// TIA Portal V20 export
TYPE "type_emRelations_em2_sequence"
// stored: Access Published, Namespace Unit1
   STRUCT
      jrOutPnPLeft : Struct
         jobs : "LAF_typeJobs";
         sequence : "LAF_typeSequence";
         selectJobStatus { S7_SetPoint := 'True'} : Array[0..10] of "LAF_typeJobStatus";
         "step" : "LER_typeStep";
         jobInterface : Struct
            stack1LoadJob2 : "LER_typeJobInterface";
            stack2LoadJob3 : "LER_typeJobInterface";
            unloadJob4 : "LER_typeJobInterface";
         END_STRUCT;
         homeCheck : Struct
            partNoDetect { ExternalWritable := 'False'} : Bool;
            partDetect { ExternalWritable := 'False'} : Bool;
         END_STRUCT;
      END_STRUCT;
      jrOutPnPRight : Struct
         jobs : "LAF_typeJobs";
         sequence : "LAF_typeSequence";
         selectJobStatus { S7_SetPoint := 'True'} : Array[0..10] of "LAF_typeJobStatus";
         "step" : "LER_typeStep";
         jobInterface : Struct
            loadJob2 : "LER_typeJobInterface";
            unloadJob3 : "LER_typeJobInterface";
         END_STRUCT;
         homeCheck : Struct
            partNoDetect { ExternalWritable := 'False'} : Bool;
            partDetect { ExternalWritable := 'False'} : Bool;
         END_STRUCT;
      END_STRUCT;
   END_STRUCT;
   // // jrOutPnPLeft."step".action1[101] : Step[101] : JOB[1] Condition
   // // jrOutPnPLeft."step".action1[110] : Step[110] : JR PP Left Clamp Open
   // // jrOutPnPLeft."step".action1[130] : Step[130] : JR PP Left Clamp Close
   // // jrOutPnPLeft."step".action1[170] : Step[170] : JR PP Left Z-Axis Wait Pos
   // // jrOutPnPLeft."step".action1[180] : Step[180] : JR PP Left X-Axis Wait Pos
   // // jrOutPnPLeft."step".action1[190] : Step[190] : JOB[1] Step End
   // // jrOutPnPLeft."step".action1[201] : Step[201] : JOB[2] Condition
   // // jrOutPnPLeft."step".action1[210] : Step[210] : JR PP Left X-Axis Loading Pos[Stack-1]
   // // jrOutPnPLeft."step".action1[211] : Step[211] : JR PP Left Z-Axis Loading Pos[Stack-1]
   // // jrOutPnPLeft."step".action1[220] : Step[220] : JR PP Left [OnPosition Unloading] => Stack #1
   // // jrOutPnPLeft."step".action1[221] : Step[221] : JR PP Left Clamp Close
   // // jrOutPnPLeft."step".action1[222] : Step[222] : JR PP Left [Request Unclamp] => Stack #1
   // // jrOutPnPLeft."step".action1[280] : Step[280] : JR PP Left X/Z-Axis Wait Pos
   // // jrOutPnPLeft."step".action1[290] : Step[290] : JOB[2] Step End
   // // jrOutPnPLeft."step".action1[301] : Step[301] : JOB[3] Condition
   // // jrOutPnPLeft."step".action1[310] : Step[310] : JR PP Left X-Axis Loading Pos[Stack-2]
   // // jrOutPnPLeft."step".action1[311] : Step[311] : JR PP left Z-Axis Loading Pos[Stack-2]
   // // jrOutPnPLeft."step".action1[320] : Step[320] : JR PP Left [OnPosition Unloading] => Stack #2
   // // jrOutPnPLeft."step".action1[321] : Step[321] : JR PP Left Clamp Close
   // // jrOutPnPLeft."step".action1[322] : Step[322] : JR PP Left [Request Unclamp] => Stack #2
   // // jrOutPnPLeft."step".action1[380] : Step[380] : JR PP Left X/Z-Axis Wait Pos
   // // jrOutPnPLeft."step".action1[390] : Step[390] : JOB[3] Step End
   // // jrOutPnPLeft."step".action1[401] : Step[401] : JOB[4] Condition
   // // jrOutPnPLeft."step".action1[410] : Step[410] : JR PP Left X-Axis Put Pos
   // // jrOutPnPLeft."step".action1[411] : Step[411] : JR PP Left Z-Axis Put Pos
   // // jrOutPnPLeft."step".action1[420] : Step[420] : JR PP Left [Unloading Ready] => Top Tape Fix Stage
   // // jrOutPnPLeft."step".action1[421] : Step[421] : JR PP Left Clamp Open
   // // jrOutPnPLeft."step".action1[422] : Step[422] : JR PP Left [Unclamp Done] => Top Tape Fix Stage
   // // jrOutPnPLeft."step".action1[480] : Step[480] : JR PP Left X/Z-Axis Wait Pos
   // // jrOutPnPLeft."step".action1[490] : Step[490] : JOB[4] Step End
   // // jrOutPnPLeft."step".transition1[101] : Step[101] : JOB[1] Condition
   // // jrOutPnPLeft."step".transition1[110] : Step[110] : JR PP Left Clamp Open
   // // jrOutPnPLeft."step".transition1[130] : Step[130] : JR PP Left Clamp Close
   // // jrOutPnPLeft."step".transition1[170] : Step[170] : JR PP Left Z-Axis Wait Pos
   // // jrOutPnPLeft."step".transition1[180] : Step[180] : JR PP Left X-Axis Wait Pos
   // // jrOutPnPLeft."step".transition1[190] : Step[190] : JOB[1] Step End
   // // jrOutPnPLeft."step".transition1[201] : Step[201] : JOB[2] Condition
   // // jrOutPnPLeft."step".transition1[210] : Step[210] : JR PP Left X-Axis Loading Pos[Stack-1]
   // // jrOutPnPLeft."step".transition1[211] : Step[211] : JR PP Left Z-Axis Loading Pos[Stack-1]
   // // jrOutPnPLeft."step".transition1[220] : Step[220] : JR PP Left [OnPosition Unloading] => Stack #1
   // // jrOutPnPLeft."step".transition1[221] : Step[221] : JR PP Left Clamp Close
   // // jrOutPnPLeft."step".transition1[222] : Step[222] : JR PP Left [Request Unclamp] => Stack #1
   // // jrOutPnPLeft."step".transition1[280] : Step[280] : JR PP Left X/Z-Axis Wait Pos
   // // jrOutPnPLeft."step".transition1[290] : Step[290] : JOB[2] Step End
   // // jrOutPnPLeft."step".transition1[301] : Step[301] : JOB[3] Condition
   // // jrOutPnPLeft."step".transition1[310] : Step[310] : JR PP Left X-Axis Loading Pos[Stack-2]
   // // jrOutPnPLeft."step".transition1[311] : Step[311] : JR PP left Z-Axis Loading Pos[Stack-2]
   // // jrOutPnPLeft."step".transition1[320] : Step[320] : JR PP Left [OnPosition Unloading] => Stack #2
   // // jrOutPnPLeft."step".transition1[321] : Step[321] : JR PP Left Clamp Close
   // // jrOutPnPLeft."step".transition1[322] : Step[322] : JR PP Left [Request Unclamp] => Stack #2
   // // jrOutPnPLeft."step".transition1[380] : Step[380] : JR PP Left X/Z-Axis Wait Pos
   // // jrOutPnPLeft."step".transition1[390] : Step[390] : JOB[3] Step End
   // // jrOutPnPLeft."step".transition1[401] : Step[401] : JOB[4] Condition
   // // jrOutPnPLeft."step".transition1[410] : Step[410] : JR PP Left X-Axis Put Pos
   // // jrOutPnPLeft."step".transition1[411] : Step[411] : JR PP Left Z-Axis Put Pos
   // // jrOutPnPLeft."step".transition1[420] : Step[420] : JR PP Left [Unloading Ready] => Top Tape Fix Stage
   // // jrOutPnPLeft."step".transition1[421] : Step[421] : JR PP Left Clamp Open
   // // jrOutPnPLeft."step".transition1[422] : Step[422] : JR PP Left [Unclamp Done] => Top Tape Fix Stage
   // // jrOutPnPLeft."step".transition1[480] : Step[480] : JR PP Left X/Z-Axis Wait Pos
   // // jrOutPnPLeft."step".transition1[490] : Step[490] : JOB[4] Step End
   // // jrOutPnPRight."step".action1[101] : Step[101] : JOB[1] Condition
   // // jrOutPnPRight."step".action1[110] : Step[110] : JR PP Right Clamp Open
   // // jrOutPnPRight."step".action1[130] : Step[130] : JR PP Right Clamp Close
   // // jrOutPnPRight."step".action1[170] : Step[170] : JR PP Right Z-Axis Wait Pos
   // // jrOutPnPRight."step".action1[180] : Step[180] : JR PP Right X-Axis Wait Pos
   // // jrOutPnPRight."step".action1[190] : Step[190] : JOB[1] Step End
   // // jrOutPnPRight."step".action1[201] : Step[201] : JOB[2] Condition
   // // jrOutPnPRight."step".action1[210] : Step[210] : JR PP Right X-Axis Loading Pos[Top Tape Fix Stage]
   // // jrOutPnPRight."step".action1[211] : Step[211] : JR PP Right Z-Axis Loading Pos[Top Tape Fix Stage]
   // // jrOutPnPRight."step".action1[220] : Step[220] : JR PP Right [Loading Ready] => Top Tape Fix Stage
   // // jrOutPnPRight."step".action1[221] : Step[221] : JR PP Right Clamp Close
   // // jrOutPnPRight."step".action1[280] : Step[280] : JR PP Right X/Z-Axis Wait Pos
   // // jrOutPnPRight."step".action1[290] : Step[290] : JOB[2] Step End
   // // jrOutPnPRight."step".action1[301] : Step[301] : JOB[3] Condition
   // // jrOutPnPRight."step".action1[310] : Step[310] : JR PP Right X-Axis Put Pos
   // // jrOutPnPRight."step".action1[311] : Step[311] : JR PP Right Z-Axis Put Pos
   // // jrOutPnPRight."step".action1[320] : Step[320] : JR PP Right [Unloading Ready] => Side Tape Fix Stage
   // // jrOutPnPRight."step".action1[321] : Step[321] : JR PP Right Clamp Open
   // // jrOutPnPRight."step".action1[322] : Step[322] : JR PP Right [Unclamp Done] => Side Tape Fix Stage
   // // jrOutPnPRight."step".action1[380] : Step[380] : JR PP Right X/Z-Axis Wait Pos
   // // jrOutPnPRight."step".action1[390] : Step[390] : JOB[3] Step End
   // // jrOutPnPRight."step".transition1[101] : Step[101] : JOB[1] Condition
   // // jrOutPnPRight."step".transition1[110] : Step[110] : JR PP Right Clamp Open
   // // jrOutPnPRight."step".transition1[130] : Step[130] : JR PP Right Clamp Close
   // // jrOutPnPRight."step".transition1[170] : Step[170] : JR PP Right Z-Axis Wait Pos
   // // jrOutPnPRight."step".transition1[180] : Step[180] : JR PP Right X-Axis Wait Pos
   // // jrOutPnPRight."step".transition1[190] : Step[190] : JOB[1] Step End
   // // jrOutPnPRight."step".transition1[201] : Step[201] : JOB[2] Condition
   // // jrOutPnPRight."step".transition1[210] : Step[210] : JR PP Right X-Axis Loading Pos[Top Tape Fix Stage]
   // // jrOutPnPRight."step".transition1[211] : Step[211] : JR PP Right Z-Axis Loading Pos[Top Tape Fix Stage]
   // // jrOutPnPRight."step".transition1[220] : Step[220] : JR PP Right [Loading Ready] => Top Tape Fix Stage
   // // jrOutPnPRight."step".transition1[221] : Step[221] : JR PP Right Clamp Close
   // // jrOutPnPRight."step".transition1[222] : Step[222] : JR PP Right [Clamp Done] => Top Tape Fix Stage
   // // jrOutPnPRight."step".transition1[280] : Step[280] : JR PP Right X/Z-Axis Wait Pos
   // // jrOutPnPRight."step".transition1[290] : Step[290] : JOB[2] Step End
   // // jrOutPnPRight."step".transition1[301] : Step[301] : JOB[3] Condition
   // // jrOutPnPRight."step".transition1[310] : Step[310] : JR PP Right X-Axis Put Pos
   // // jrOutPnPRight."step".transition1[311] : Step[311] : JR PP Right Z-Axis Put Pos
   // // jrOutPnPRight."step".transition1[320] : Step[320] : JR PP Right [Unloading Ready] => Side Tape Fix Stage
   // // jrOutPnPRight."step".transition1[321] : Step[321] : JR PP Right Clamp Open
   // // jrOutPnPRight."step".transition1[322] : Step[322] : JR PP Right [Unclamp Done] => Side Tape Fix Stage
   // // jrOutPnPRight."step".transition1[380] : Step[380] : JR PP Right X/Z-Axis Wait Pos
   // // jrOutPnPRight."step".transition1[390] : Step[390] : JOB[3] Step End
END_TYPE
